Staubli VAL3: remSetIPVals.pgx

program remSetIPVals(string& sArgs[] (dimensions=1), string& sReturn[] (dimensions=1))
  local bool bOk
  local num nArg
  local num nIP
  local num nTemp
  local trsf trIP
begin
  // Change the values of the active interaction point.
  //
  // Arguments are "X Y Z RX RY RZ"
  //
  logMsg("call remSetIPVals")
  nArg=0
  trIP={0,0,0,0,0,0}
  while nArg<7
    sArgs=toNum(sArgs,nTemp,bOk)
    if bOk
      switch nArg
        case 0
          nIP=nTemp
        break
        case 1
          trIP.x=nTemp
        break
        case 2
          trIP.y=nTemp
        break
        case 3
          trIP.z=nTemp
        break
        case 4
          trIP.rx=nTemp
        break
        case 5
          trIP.ry=nTemp
        break
        case 6
          trIP.rz=nTemp
        break
      endSwitch
      nArg=nArg+1
    else
      call remErrNum("SETIPVALS",sArgs,sReturn)
      return
    endIf
  endWhile
  if nIP==0
    fIP1.trsf=trIP
  else
    fIP2.trsf=trIP
  endIf
  sReturn="SETIPVALS"
end
